{attribute addProperty BoxType "EK1100-0000-0018"}
{attribute addProperty Id "A_0016_BK1250_0000_0017A_0016_BK1250_0000_0017_446ACE0300"}
{attribute addProperty CRC "1155270411"}
{attribute addProperty SizeInBites "0"}
{attribute addProperty SizeInBytes "0"}
TYPE Term_474_EK1100_44DC070B EXTENDS EK1100_179A0949 :
STRUCT
	{attribute addProperty Name "A_0016_BK1250_0000_0017"}
	A_0016_BK1250_0000_0017 : A_0016_BK1250_0000_0017_446ACE03;
END_STRUCT
END_TYPE

(* stored: Version 1.2.0.0, ProductVersion 3.1.4024.9
   DUT Term_474_EK1100_44DC070B: Id {3cf5450f-e073-4c38-8d21-cd51f4b41e3c} *)
